// TIA Portal V20 export
FUNCTION_BLOCK "Simulation"   // FB105, LAD
// stored: MemoryReserve 100, Namespace Unit1.Em4, SetENOAutomatically false
   VAR
      Simulation_addon_Instance { S7_SetPoint := 'True'} : "Simulation_addon";
   END_VAR
BEGIN

REGION Network 1: cmFeederCylinderUpDown
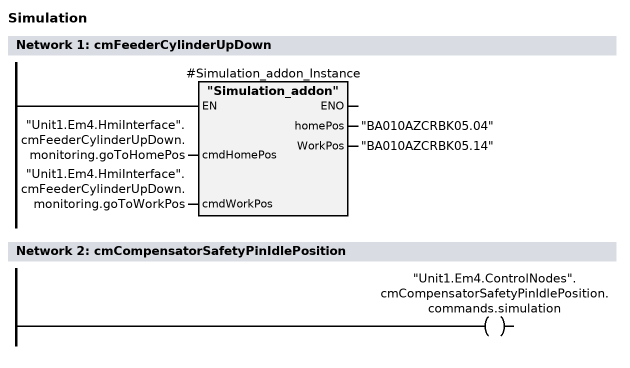
   RUNG wire#powerrail
      #Simulation_addon_Instance(cmdHomePos := "Unit1.Em4.HmiInterface".cmFeederCylinderUpDown.monitoring.goToHomePos, cmdWorkPos := "Unit1.Em4.HmiInterface".cmFeederCylinderUpDown.monitoring.goToWorkPos, homePos => "BA010AZCRBK05.04", WorkPos => "BA010AZCRBK05.14")
   END_RUNG
   // the same network as SCL:
   #Simulation_addon_Instance(cmdHomePos := "Unit1.Em4.HmiInterface".cmFeederCylinderUpDown.monitoring.goToHomePos,   // "Simulation_addon"
                           cmdWorkPos := "Unit1.Em4.HmiInterface".cmFeederCylinderUpDown.monitoring.goToWorkPos,
                           homePos => "BA010AZCRBK05.04",
                           WorkPos => "BA010AZCRBK05.14");
END_REGION

REGION Network 2: cmCompensatorSafetyPinIdlePosition
   RUNG wire#powerrail
      Coil( "Unit1.Em4.ControlNodes".cmCompensatorSafetyPinIdlePosition.commands.simulation )
   END_RUNG
   // the same network as SCL:
   "Unit1.Em4.ControlNodes".cmCompensatorSafetyPinIdlePosition.commands.simulation := TRUE;
END_REGION
END_FUNCTION_BLOCK
